// TIA Portal V18 export
DATA_BLOCK "HeatingPLC_vAI_Vars"   // DB11001
{ S7_Optimized_Access := 'FALSE' }
VERSION : 0.1
// stored: AutoNumber false, DBAccessibleFromOPCUA true, IsOnlyStoredInLoadMemory false, IsWriteProtectedInAS false
   VAR
      vAI1 { S7_SetPoint := 'True'} : "UDT_vAI";
      vAI2 { S7_SetPoint := 'True'} : "UDT_vAI";
      vAI3 { S7_SetPoint := 'True'} : "UDT_vAI";
      vAI4 { S7_SetPoint := 'True'} : "UDT_vAI";
      vAI5 { S7_SetPoint := 'True'} : "UDT_vAI";
      vAI6 { S7_SetPoint := 'True'} : "UDT_vAI";
      vAI7 { S7_SetPoint := 'True'} : "UDT_vAI";
      vAI8 { S7_SetPoint := 'True'} : "UDT_vAI";
      vAI9 { S7_SetPoint := 'True'} : "UDT_vAI";
      vAI10 { S7_SetPoint := 'True'} : "UDT_vAI";
      vAI11 { S7_SetPoint := 'True'} : "UDT_vAI";
      vAI12 { S7_SetPoint := 'True'} : "UDT_vAI";
      vAI13 { S7_SetPoint := 'True'} : "UDT_vAI";
      vAI14 { S7_SetPoint := 'True'} : "UDT_vAI";
      vAI15 { S7_SetPoint := 'True'} : "UDT_vAI";
      vAI16 { S7_SetPoint := 'True'} : "UDT_vAI";
   END_VAR
BEGIN
   vAI1.rValue := 0.0;
   vAI1.rMax := 2000.0;
   vAI1.iFuncSystemID := 2;
   vAI1.iFuncVar := 1;
   vAI2.rValue := 22.0;
   vAI2.rMin := -25.0;
   vAI2.rMax := 25.0;
   vAI2.iFuncSystemID := 1;
   vAI2.iFuncVar := 2;
   vAI3.rValue := 21.0;
   vAI3.rMin := -25.0;
   vAI3.rMax := 25.0;
   vAI3.iFuncSystemID := 2;
   vAI3.iFuncVar := 2;
   vAI4.rValue := 19.0;
   vAI4.rMax := 1000.0;
   vAI4.iFuncSystemID := 1;
   vAI4.iFuncVar := 1;
   vAI5.rValue := 21.0;
   vAI5.rMax := 1000.0;
   vAI5.iFuncSystemID := 1;
   vAI5.iFuncVar := 14;
   vAI6.iFuncSystemID := 0;
   vAI6.iFuncVar := 0;
   vAI9.rValue := 665.0;
   vAI9.iFuncSystemID := 0;
   vAI9.iFuncVar := 0;
   vAI10.rValue := 21.1;
   vAI10.iFuncSystemID := 0;
   vAI10.iFuncVar := 0;
   vAI11.rValue := 21.5;
   vAI11.iFuncSystemID := 0;
   vAI11.iFuncVar := 0;
   vAI12.rValue := 18.8;
   vAI12.iFuncSystemID := 0;
   vAI12.iFuncVar := 0;
   vAI13.rValue := 22.6;
   vAI13.iFuncSystemID := 0;
   vAI13.iFuncVar := 0;
   vAI14.rValue := 45.0;
   vAI14.iFuncSystemID := 0;
   vAI14.iFuncVar := 0;
END_DATA_BLOCK
